{attribute 'qualified_only'}
VAR_GLOBAL
	Reset AT %Q*: BOOL;
	Run AT %Q*: BOOL;
	iReset AT %I*: BOOL;
	
	Estop_ok AT %I*: BOOL;
	ECU1_2_Ok AT %I*: BOOL;
	CBU_LB_Ok AT %I*: BOOL;
	MCS_OK AT %I*: BOOL;
	
END_VAR

(* stored: Version 1.1.0.1, ProductVersion 3.1.4024.14
   GVL Safety_Tags: Id {a36fc3c1-26ca-4ca9-8fbb-6959cc4e5ca4} *)
